TYPE ST_CFG_LiftTableEmulation :
STRUCT
	PositionUp 		: INT := 500;
	PositionDown 	: INT := 100;
END_STRUCT
END_TYPE

(* stored: Version 1.1.0.1, ProductVersion 3.1.4024.9
   DUT ST_CFG_LiftTableEmulation: Id {56ef6d7d-9bba-441e-a76e-98b5ea84f219} *)
